# EPICS autosave request: 3-6/GalilSup/Db/galil_motor_settings.req
$(P)$(M).MDEL
$(P)$(M).ADEL
